// TIA Portal V16 export
// export: Created 2022-11-17T15:49:31.3412389Z, ExportSetting WithDefaults, DisplayName Totally Integrated Automation Portal, DisplayVersion V16 Update 6, DisplayName TIA Portal Version Control Interface, DisplayVersion V16 Update 2, DisplayName TIA Portal Openness, DisplayVersion V16 Update 6, DisplayName SINAMICS Startdrive Advanced, DisplayVersion V16 Update 5, DisplayName SINAMICS Startdrive G130, G150, S120, S150, SINAMICS MV, S210, DisplayVersion V16 Update 5, DisplayName SINAMICS Startdrive G110M, G120, G120C, G120D, G120P, G115D, DisplayVersion V16 Update 5, DisplayName STEP 7 Professional, DisplayVersion V16 Update 6, DisplayName STEP 7 Safety, DisplayVersion V16, DisplayName WinCC Advanced, DisplayVersion V16 Update 6
FUNCTION "FC101_AxisPositioningRev" : Void   // FC101, LAD
TITLE = Axis positioning
{ S7_Optimized_Access := 'FALSE' }
AUTHOR : Robopac
VERSION : 0.0
// stored: AutoNumber false, IsIECCheckEnabled false, SetENOAutomatically false, UDAEnableTagReadback false
   VAR_INPUT
      Start : Bool;   // Start dell'asse
      ExtraAvanti : Bool;   // Sensore di extracorsa avanti
      ExtraIndietro : Bool;   // Sensore di extracorsa indietro
      PosAttuale : Int;   // Posizione attuale dell'asse
      PosDest : Int;   // Posizione di destinazione dell'asse
      Dec : Int;   // Decelerazione
      H_Isteresi : Int;   // Isteresi
   END_VAR
   VAR_OUTPUT
      VelBassa : Bool;   // Asse all'interno dell'intervallo di decelerazione
      Avanti : Bool;   // Asse avanti
      Indietro : Bool;   // Asse indietro
   END_VAR
   VAR_IN_OUT
      PosOk : Bool;   // Asse in posizione
   END_VAR
   VAR_TEMP
      PosDestMenoH : Int;   // Posizione di destinazione asse-Isteresi
      PosDestPiuH : Int;   // Posizione di destinazione asse+Isteresi
      PosDestMenoDec : Int;   // Posizione di destinazione asse-Decelerazione
      PosDestPiuDec : Int;   // Posizione di destinazione asse+Decelerazione
   END_VAR
   VAR_TEMP   // added for the SCL form of the ladder/FBD networks
      _w1 : Bool;
   END_VAR
BEGIN

REGION Network 1
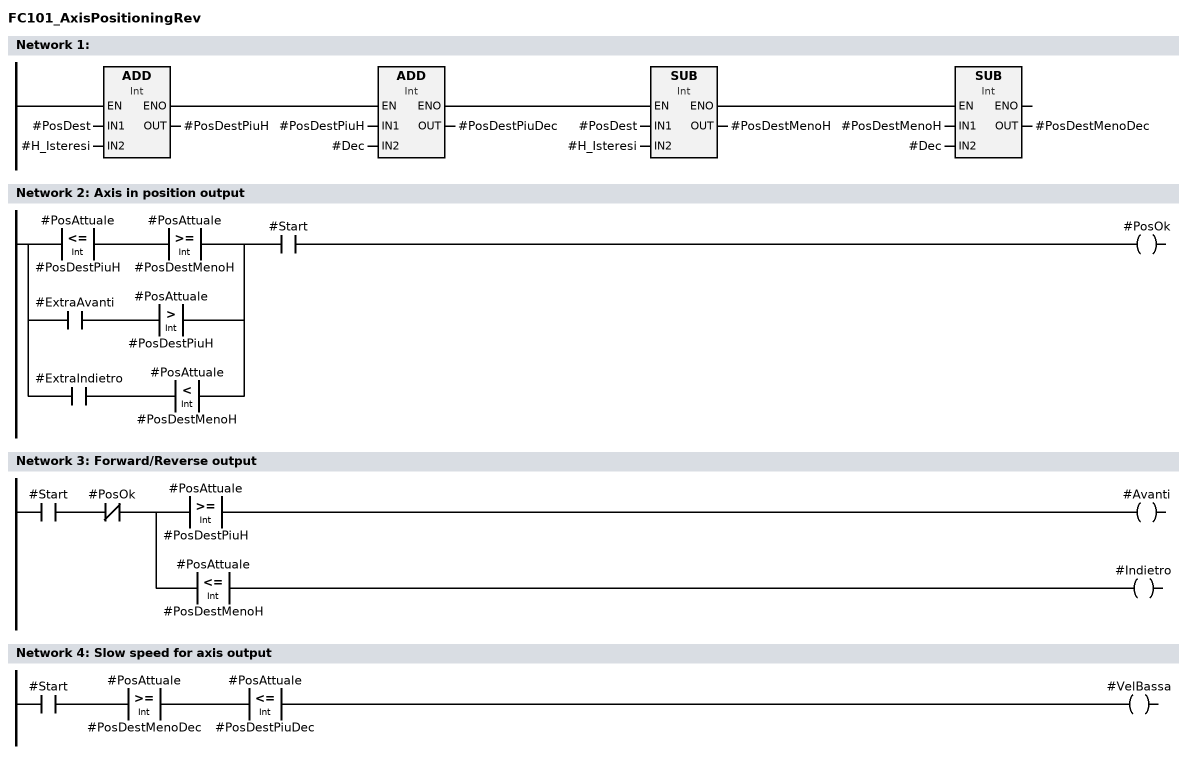
   RUNG wire#powerrail
      { S7_Templates := "SrcType := Int"; S7_GenerateENO := "TRUE" } Add(in1 := #PosDest, in2 := #H_Isteresi, out => #PosDestPiuH)
      { S7_Templates := "SrcType := Int"; S7_GenerateENO := "TRUE" } Add(in1 := #PosDestPiuH, in2 := #Dec, out => #PosDestPiuDec)
      { S7_Templates := "SrcType := Int"; S7_GenerateENO := "TRUE" } Sub(in1 := #PosDest, in2 := #H_Isteresi, out => #PosDestMenoH)
      { S7_Templates := "SrcType := Int"; S7_GenerateENO := "TRUE" } Sub(in1 := #PosDestMenoH, in2 := #Dec, out => #PosDestMenoDec)
   END_RUNG
   // the same network as SCL:
   // ENO of a box is taken as its EN; it also drops when the box reports an error
   #PosDestPiuH := #PosDest + #H_Isteresi;
   #PosDestPiuDec := #PosDestPiuH + #Dec;
   #PosDestMenoH := #PosDest - #H_Isteresi;
   #PosDestMenoDec := #PosDestMenoH - #Dec;
END_REGION

REGION Network 2: Axis in position output
   RUNG wire#powerrail
      { S7_Templates := "SrcType := Int" } LE_Contact(in1 := #PosAttuale, in2 := #PosDestPiuH)
      { S7_Templates := "SrcType := Int" } GE_Contact(in1 := #PosAttuale, in2 := #PosDestMenoH)
      wire#w1
      Contact( #Start )
      Coil( #PosOk )
   END_RUNG
   RUNG wire#powerrail
      Contact( #ExtraAvanti )
      { S7_Templates := "SrcType := Int" } GT_Contact(in1 := #PosAttuale, in2 := #PosDestPiuH)
   END_RUNG wire#w1
   RUNG wire#powerrail
      Contact( #ExtraIndietro )
      { S7_Templates := "SrcType := Int" } LT_Contact(in1 := #PosAttuale, in2 := #PosDestMenoH)
   END_RUNG wire#w1
   // the same network as SCL:
   #PosOk := (((#PosAttuale <= #PosDestPiuH) AND (#PosAttuale >= #PosDestMenoH)) OR (#ExtraAvanti AND (#PosAttuale > #PosDestPiuH)) OR (#ExtraIndietro AND (#PosAttuale < #PosDestMenoH))) AND #Start;
END_REGION

REGION Network 3: Forward/Reverse output
   RUNG wire#powerrail
      Contact( #Start )
      I_Contact( #PosOk )
      wire#w1
      { S7_Templates := "SrcType := Int" } GE_Contact(in1 := #PosAttuale, in2 := #PosDestPiuH)
      Coil( #Avanti )
   END_RUNG
   RUNG wire#w1
      { S7_Templates := "SrcType := Int" } LE_Contact(in1 := #PosAttuale, in2 := #PosDestMenoH)
      Coil( #Indietro )
   END_RUNG
   // the same network as SCL:
   #_w1 := #Start AND NOT #PosOk;
   #Avanti := #_w1 AND (#PosAttuale >= #PosDestPiuH);
   #Indietro := #_w1 AND (#PosAttuale <= #PosDestMenoH);
END_REGION

REGION Network 4: Slow speed for axis output
   RUNG wire#powerrail
      Contact( #Start )
      { S7_Templates := "SrcType := Int" } GE_Contact(in1 := #PosAttuale, in2 := #PosDestMenoDec)
      { S7_Templates := "SrcType := Int" } LE_Contact(in1 := #PosAttuale, in2 := #PosDestPiuDec)
      Coil( #VelBassa )
   END_RUNG
   // the same network as SCL:
   #VelBassa := #Start AND (#PosAttuale >= #PosDestMenoDec) AND (#PosAttuale <= #PosDestPiuDec);
END_REGION
END_FUNCTION
